FUNCTION F_Toggle : BOOL
VAR_INPUT
END_VAR
VAR
	
END_VAR

END_FUNCTION

(* stored: Version 1.1.0.1, ProductVersion 3.1.4024.16
   POU F_Toggle: Id {08f9f8cb-49e7-4dc8-bd61-530aee0ec112}, SpecialFunc None *)
